DATA_BLOCK "dbArchiveAutoRectifier"
{ S7_Optimized_Access := 'TRUE' }
VERSION : 0.8
NON_RETAIN
"fbArchiveAutoRectifier"

BEGIN

END_DATA_BLOCK

